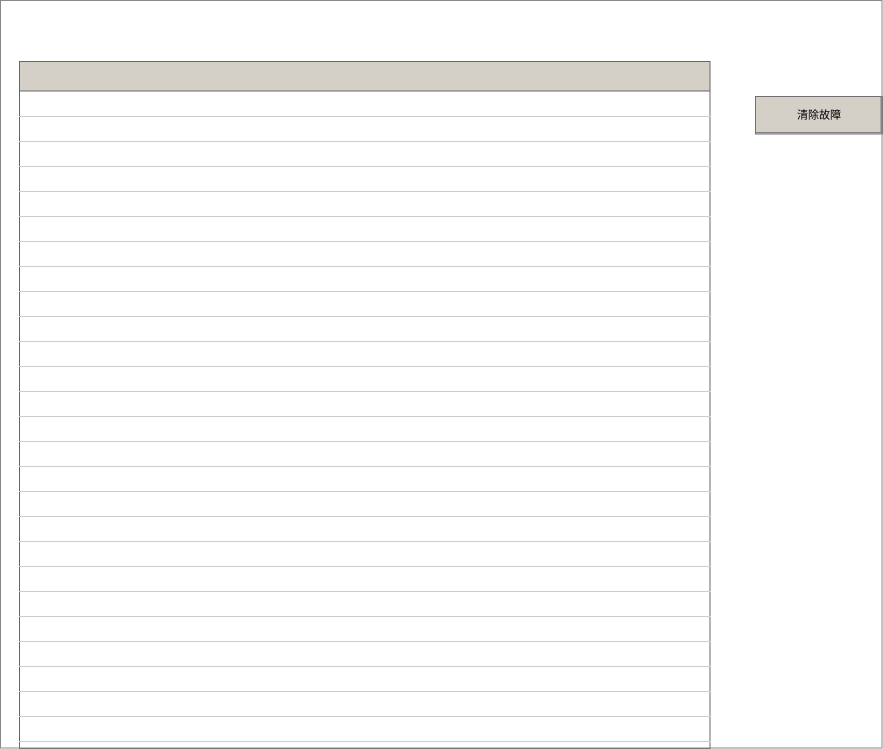
VISUALIZATION arm2SafetyCheck  // 883x749
    Table (19,61 691x688), data array: g_ArrayErrCodeTypeTest[2]
        p3854506369: g_ArrayErrCodeTypeTest[2][1][INDEX]
        p1892666644: g_ArrayErrCodeTypeTest[2][2][INDEX]
        p338671338: g_ArrayErrCodeTypeTest[3][INDEX]
        p2170511999: g_ArrayErrCodeTypeTest[4][INDEX]
        p3723444502: g_ArrayErrCodeTypeTest[5][INDEX]
    Button (755,96 128x38), "清除故障", colour toggle: g_clearFault
        tap g_clearFault
END_VISUALIZATION

(* stored: Version 1.1.0.1, ProductVersion 3.1.4024.11
   Visu arm2SafetyCheck: Id {40f10079-ccd2-4736-bb3e-31310460190e} *)
